// TIA Portal V20 export
VAR_GLOBAL   // PLC tag table "PLC_Centralizer_PLC_Production_And_Rework"
   In AT %I500.0 : "IO_Device_Inputs";
   Out AT %Q500.0 : "IO_Device_Outputs";
END_VAR
